METHOD mxGetMk5sData : BOOL
VAR_INPUT
	bItemNumber	: BYTE;
	pstrSetting	: POINTER TO Mk5s_Display_Helpers_Interfaces.strProtectionInfo_v2;
	xSavedData	: BOOL;
END_VAR
VAR_OUTPUT
	bAccesLevelDisplay	: BYTE := _FLAG_Acces_User;
	bAccesLevelEdit	: BYTE := _FLAG_Acces_User;
	xNoEditing	: BOOL := FALSE;
	xNoDisplay	: BOOL := FALSE;
END_VAR
CASE bItemNumber OF
	1:	pstrSetting^.eType := ENUM_VALUE_TYPE.analog;
		pstrSetting^.wTIDName := gTxt_COMITEM_104;
		pstrSetting^.strItem.diValue := itfSTCValve.prpwError;
		xNoDisplay := pstrSetting^.strItem.diValue = 0;
		mxGetMk5sData := TRUE;
ELSE
		mxGetMk5sData := FALSE;
END_CASE
END_METHOD

METHOD mxSetMk5sData : BOOL
VAR_INPUT
	bItemNumber	: BYTE;
	diValue	: DINT;
END_VAR
VAR_OUTPUT
	wSDO	: WORD;
	bSI	: BYTE;
	dataODItem	: Mk5s_Display_Helpers_Interfaces._DEFINITIONS_.ODItem;
	xEditValueSuccessful	: BOOL;
END_VAR
mxSetMk5sData := TRUE;
END_METHOD

METHOD mInit
VAR_INPUT
	itfSTCValveIn	: itf_STCValve;
END_VAR
itfSTCValve := itfSTCValveIn;
END_METHOD

END_FUNCTION_BLOCK

// Aorta/AortaEngine/fbtAortaEngine_Base
FUNCTION_BLOCK fbtAortaEngine_Base IMPLEMENTS itf_STCValve
VAR
	xActive						 : BOOL;
	xActivePI					 : BOOL;	
	bNumberSTC					 : BYTE;
	xCheckCAN					 : BOOL := TRUE;
	xEnergyRecoveryActive		 : BOOL := FALSE;
	itfEnergyRecoveryRegulation  : itf_EnergyRecoveryRegulation;
	bAbsoluteOffset				 : BYTE := 127;
	
	itfIData_PI				: itf_InternalValue_PI;

	fbAorta_Trinamics		: fbtAorta_Trinamics; 
	fbSettingsDownloader 	: fbtAortaSettingsDownloader;
	
	eStateMain				: ENUM_AortaEngine_StateMain;
	eStateHoming			: ENUM_AortaEngine_StateHoming;
	eStateOperating			: ENUM_AortaEngine_StateOperating;
	eStateRetract			: ENUM_AortaEngine_StateRetract;
	
	wEnableErrorCount		: WORD;
	wResetCount				: WORD;
	
	itfLocalRoot			: itf_SystemRoot;
	
	itfWarmUpTemperature		: itf_BaseIO;
	rsWarmUp					: RS;

	itfPositionInput			: itf_BaseIO;
	itfPositionOutput			: itf_BaseIO;
	
	wSDO_STCValve				: WORD;
	
	fbIVL_ActualPosition		: fbtIVL_STCPosition;
	fbIVL_RequiredPosition		: fbtIVL_STCPosition;
	
	fbSTCValve_Protection		: fbtProtecSpec_STCValve;
	
	tFixedPositionTimeoutTime	: TIME;	
	wRangeOffsetLower			: WORD;
	wRangeOffsetUpper			: WORD;
	wWorkingRange				: WORD;
	
	xStart						: BOOL;
	xStartHoming				: BOOL;
	xStartPosition				: BOOL;
	xStartRetract				: BOOL;
	CycleTime 					: TON;

	odError						: ODItem;
	dwStroke_MicroSteps			: DWORD;
	dwStroke_FullSteps			: DWORD;
	rStroke_Rotations			: REAL;
	
	// Settings
	wCycleTime				: WORD;
	wPositioningTimeOut		: WORD;
	wHomingTimeOut			: WORD;

	tInitiateRetryDelayTime		: TIME;
	bMaxHomingRetries			: BYTE;
	bHomingRetries				: BYTE;
	tHomeAgainDelayTime			: TIME;
	tonHomeAgainDelay			: TON;
	dwErrorPosition				: DWORD;
	dwMicroStepsInMove			: DWORD;
	wRetractRange				: WORD;
	wMinimumFullStepRange		: WORD;
	
	diPosition					: DINT;
	dwPositionPrev				: DWORD;
	bFirstWarmUpTemperature		: BYTE;
	wRangeOffsetLowerMargin		: WORD;
	

	iPositionInputRangeMin		: INT;
	iPositionInputRangeMax		: INT;
	iPositionOutputRangeMin		: INT;
	iPositionOutputRangeMax		: INT;
	iPositionOutput				: INT;
	
	itfHomings					: itf_Counter;
    itfStalls					: itf_Counter;
	itfRotations				: itf_Counter;
	
	internalRotationsCounter	: DWORD;
	
	xStartForcedHoming	: BOOL;
	xHomingActive	: BOOL;
	xFixedPositionActive	: BOOL;
	tonFixedPositionTimeout	: TON;

	diPositionInOffState	: DINT;
		
	itfRetainStatus				:itf_Retain_3000_X;
	
	awAlarmNames									: ARRAY[1..6] OF WORD := [gTxt_Alarm_13453, gTxt_Alarm_13454, gTxt_Alarm_13455, gTxt_Alarm_13456, gTxt_Alarm_13457, gTxt_Alarm_13458];
	awAlarmSDOs										: ARRAY[1..6] OF WORD := [16#2815, 16#2895, 16#2896, 16#2897, 16#2898, 16#2899];
	
	awSTCValveHomingCycles							: ARRAY[1..6] OF WORD := [13459, 13460, 13461, 13462, 13463, 13464];
	awSTCValveStalls								: ARRAY[1..6] OF WORD := [13465, 13466, 13467, 13468, 13469, 13470];
	awSTCValveRotations								: ARRAY[1..6] OF WORD := [13471, 13472, 13473, 13474, 13475, 13476];
	
	
	// Debug
	adi_Testing					: ARRAY[1..9] OF DINT;
	diDebugError				: DINT;
	diDebugErrorPosition		: DINT;
	diDebugMicroStepsInMove		: DINT;
	diDebugPosition				: DINT;
	diDebugRotDirection			: DINT;
	diDebugStroke_FullSteps		: DINT;
	diDebugStroke_MicroSteps	: DINT;
	diDebugStroke_Rotations		: DINT;
	diDebugStallDetectPosition	: DINT;
	diDebugStallRetractPosition	: DINT;
	diDebugRetractDelta			: DINT;
	diDebugStatusWord			: DINT;
	diDebugError11Counter		: DINT;
	diDebug_numberStalls		: DINT;
	xDebug_ok					: BOOL;
	wDebugError2				: WORD;

END_VAR

METHOD mxInit_SysPyLog : BOOL
VAR_INPUT
END_VAR
SysPyLog.mxAdd(eCode := eLogCodes._fixed_1, pData := ADR(xDebug_ok),sNaam := 'xOk', eType := eLogTypes._byte);
SysPyLog.mxAdd(eCode := eLogCodes._fixed_1, pData := ADR(odError.wValue[1]),sNaam := 'Aorta Error', eType := eLogTypes._word);
SysPyLog.mxAdd(eCode := eLogCodes._fixed_1, pData := ADR(wDebugError2),sNaam := 'Aorta Error2', eType := eLogTypes._word);
SysPyLog.mxAdd(eCode := eLogCodes._fixed_1, pData := ADR(eStateMain),sNaam := 'State Main', eType := eLogTypes._byte);
SysPyLog.mxAdd(eCode := eLogCodes._fixed_1, pData := ADR(eStateOperating),sNaam := 'State Operating', eType := eLogTypes._byte);
SysPyLog.mxAdd(eCode := eLogCodes._fixed_1, pData := ADR(eStateHoming),sNaam := 'State Homing', eType := eLogTypes._byte);
SysPyLog.mxAdd(eCode := eLogCodes._fixed_1, pData := ADR(diDebugStroke_FullSteps),sNaam := 'Full steps stroke', eType := eLogTypes._byte);
SysPyLog.mxAdd(eCode := eLogCodes._fixed_1, pData := ADR(diDebugErrorPosition),sNaam := 'Error Position', eType := eLogTypes._dint);
SysPyLog.mxAdd(eCode := eLogCodes._fixed_1, pData := ADR(diDebugMicroStepsInMove),sNaam := 'Micro Steps In Move', eType := eLogTypes._dint);
SysPyLog.mxAdd(eCode := eLogCodes._fixed_1, pData := ADR(diDebugRotDirection),sNaam := 'Rotation Direction', eType := eLogTypes._dint);
SysPyLog.mxAdd(eCode := eLogCodes._fixed_1, pData := ADR(diDebugStroke_FullSteps),sNaam := 'Stroke In Full Steps', eType := eLogTypes._dint);
SysPyLog.mxAdd(eCode := eLogCodes._fixed_1, pData := ADR(diDebug_numberStalls),sNaam := 'Number of Stalls', eType := eLogTypes._dint);
END_METHOD

METHOD mxInit : BOOL
VAR_INPUT
	wSDOIn			: WORD;
	itfEnergyRecoveryRegulationIn : itf_EnergyRecoveryRegulation;
END_VAR
VAR
	TmpItem	: ODItem;		
	itfLookupTables	: itf_lookuptables;
	itfCounters		: itf_Counters;
END_VAR
mxInit := TRUE;
xActive := TRUE;

IF NOT __QUERYINTERFACE(GVL_itfRoot,	itfLocalRoot) THEN	mxInit := FALSE;	RETURN;	END_IF

IF NOT CmpODRead(wSDO_STCValve,	27,	ADR(TmpItem))  THEN
	xActive := FALSE;
	fbIVL_ActualPosition.prpxDataBaseDefined 	:= FALSE;
	fbIVL_RequiredPosition.prpxDataBaseDefined  := FALSE;
	RETURN;
END_IF

IF TmpItem.bValue[3] = 0 THEN
	xActive := FALSE;
END_IF

itfCounters					:= itfLocalRoot.prpitfCounters;
itfLocalRoot.prpitfRetain.mxGetRetainPrimaryMachine(itfRetainPrimaryMachineStatus=>itfRetainStatus);
itfLocalRoot.prpitfCANtainer.mxAttachDriver(eType := eTypeDrivers.AortaDrives, itfcanopendriver := fbAorta_Trinamics.prpitfCANOpenDriver);
itfLocalRoot.prpitfCANtainer.mxAttachDownloader(itfsettingsdownloader := fbSettingsDownloader);
itfLookupTables				:= itfLocalRoot.prpitfLookupTables;

IF		itfLookupTables	= 0 OR	itfCounters	= 0 OR itfRetainStatus = 0 THEN	
	mxInit := FALSE;	RETURN;	END_IF

itfHomings		:= itfCounters.mitfGetCounter(awSTCValveHomingCycles[bNumberSTC]);
itfStalls		:= itfCounters.mitfGetCounter(awSTCValveStalls[bNumberSTC]);
itfRotations	:= itfCounters.mitfGetCounter(awSTCValveRotations[bNumberSTC]);

mxInit := mxInit AND mxLoadSettings(itfEnergyRecoveryRegulationIn); 

xStart := TRUE;
eStateMain := ENUM_AortaEngine_StateMain.Enable;
wEnableErrorCount := 0;
wResetCount := 0;

fbAorta_Trinamics.mxInit(bCANAddress := 6 ,wHomingTimeOutIn := wHomingTimeOut ,wPositioningTimeOutIn :=wPositioningTimeOut );
fbSettingsDownloader.mxInit(ADR(fbAorta_Trinamics));

// Initialising STC Valve Alarm
mxInit := mxInit AND fbSTCValve_Protection.mxInitSpecial(wNameIn := awAlarmNames[bNumberSTC], wSDOIn := awAlarmSDOs[bNumberSTC], THIS^);

mxInit_SysPyLog();
END_METHOD

METHOD mxInit_Output : BOOL
VAR_INPUT
	bNumberSTCIn			: BYTE;
	wSDOIn					: WORD;
	wMPL_actualPosition		: WORD;
	wMPL_requiredPosition	: WORD;
	wName_actualPosition	: WORD;
	wName_requiredPosition	: WORD;
END_VAR
VAR
	itfLookupTables	: itf_lookuptables;
END_VAR
mxInit_Output := TRUE;
bNumberSTC := bNumberSTCIn;
wSDO_STCValve := wSDOIn;
mxInit_Output := mxInit_Output AND fbIVL_ActualPosition.mxInit(wMPL_actualPosition);
mxInit_Output := mxInit_Output AND fbIVL_RequiredPosition.mxInit(wMPL_requiredPosition);
END_METHOD

METHOD mxLoadSettings : BOOL
VAR_INPUT
	itfEnergyRecoveryRegulationIn : itf_EnergyRecoveryRegulation;
END_VAR
VAR
	TmpItem						  : ODItem;
	tFixedPositionTimeoutTimeUnit : ENUM_TimeUnit;
	i							  : BYTE;
	itfIData_temp				  : itf_InternalValue;
END_VAR
// Collect Data
mxLoadSettings := TRUE;

FOR i := 1 TO 11 BY 1 DO //see Hi5 SDO 2666
    CmpODRead(ENUM_SDO_2000.Aorta, i ,ADR(TmpItem));

	CASE i OF
		
	1: 
		tInitiateRetryDelayTime		:= TmpItem.bValue[1] * T#1S;
		bMaxHomingRetries			:= TmpItem.bValue[2];
		tHomeAgainDelayTime			:= TmpItem.bValue[3] * T#1H;
		wHomingTimeOut 				:= TmpItem.bValue[4];
	
	2:
		wRetractRange			:= TmpItem.wValue[1];
		wMinimumFullStepRange	:= TmpItem.wValue[2];
	
	3:
	
		wRangeOffsetLower	:= TmpItem.wValue[1];
		wCycleTime 			:= TmpItem.wValue[2];
		
	4:
		wPositioningTimeOut := TmpItem.wValue[1];
		IF TmpItem.wValue[2] = 0 THEN mxLoadSettings:= FALSE; RETURN; END_IF; 
		itfLocalRoot.prpitfLookupTables.prpitfIVLList.mxFind(wFind:=TmpItem.wValue[2], itfFound=>itfIData_temp);  
		IF NOT __QUERYINTERFACE(itfIData_temp,	itfIData_PI) THEN	mxLoadSettings := FALSE;	RETURN;	END_IF 
		mxLoadSettings:=mxLoadSettings AND itfIData_PI<>0;
		
	5:
		wRangeOffsetUpper	:= GVL_Aorta.wControlRange - TmpItem.wValue[1];
		IF itfPositionOutput <> 0 THEN
			itfLocalRoot.prpitfLookupTables.prpitfMPLList.mxFind(wFind:=TmpItem.wValue[2], itfFound=>itfPositionOutput);
			mxLoadSettings:=mxLoadSettings AND itfPositionOutput<>0;	
		END_IF
		
			
	9:
		wRangeOffsetLowerMargin	:= TmpItem.wValue[1];
		bFirstWarmUpTemperature	:= TmpItem.bValue[3];
	
	10:
		IF TmpItem.wValue[2] <> 0 THEN
			itfLocalRoot.prpitfLookupTables.prpitfMPLList.mxFind(wFind:=TmpItem.wValue[2], itfFound=>itfPositionInput);
			mxLoadSettings:=mxLoadSettings AND itfPositionInput<>0;
		END_IF
		
		
	11:
		IF TmpItem.wValue[1] = 0 THEN mxLoadSettings:= FALSE; RETURN; END_IF; 
		itfLocalRoot.prpitfLookupTables.prpitfMPLList.mxFind(wFind:=TmpItem.wValue[1], itfFound=>itfWarmUpTemperature);
		mxLoadSettings:=mxLoadSettings AND itfWarmUpTemperature<>0;

	ELSE
		IF NOT (i = 6 OR i = 7 OR i = 8) THEN
			mxLoadSettings := FALSE;	
		END_IF
	END_CASE
END_FOR

CmpODRead(ENUM_SDO_2000.Aorta,	23,	ADR(TmpItem));
tFixedPositionTimeoutTimeUnit := TmpItem.bValue[3];
xEnergyRecoveryActive		  := BYTE_TO_BOOL(TmpItem.bValue[2]);

CASE tFixedPositionTimeoutTimeUnit OF
	ENUM_TimeUnit.Millisecond	: tFixedPositionTimeoutTime := TmpItem.bValue[4] * T#1MS;
	ENUM_TimeUnit.Second	: tFixedPositionTimeoutTime := TmpItem.bValue[4] * T#1S;
	ENUM_TimeUnit.Minute	: tFixedPositionTimeoutTime := TmpItem.bValue[4] * T#1M;
	ENUM_TimeUnit.Hour	: tFixedPositionTimeoutTime := TmpItem.bValue[4] * T#1H;
	ENUM_TimeUnit.Day	: tFixedPositionTimeoutTime := TmpItem.bValue[4] * T#1D;
END_CASE

wWorkingRange	:= wRangeOffsetUpper - wRangeOffsetLower;

IF xEnergyRecoveryActive = 1 THEN
	mxLoadSettings := mxLoadSettings AND CmpODRead(_wSDO2_EnergyRecoveryRegulation, 1, ADR(TmpItem));
	itfEnergyRecoveryRegulation := itfEnergyRecoveryRegulationIn;
	mxLoadSettings := mxLoadSettings AND itfEnergyRecoveryRegulation <> 0;
END_IF

CmpODRead(ENUM_SDO_2000.Aorta,	35,	ADR(TmpItem));	
	diPositionInOffState:=TmpItem.diValue;
END_METHOD

METHOD mxRun : BOOL
VAR
	wError	: WORD;
	bError  : BYTE;
	xOk		: BOOL;
	xSwitchToER		: BOOL;
END_VAR
IF NOT xActive THEN
	RETURN;
END_IF

//  fbAorta_Trinamics.mxRun(); running via CANTainer
IF (fbAorta_Trinamics.mxConfigurationError(bError => bError) OR THIS^.prpxCANDriverError) AND xCheckCAN THEN
	eStateMain	:= ENUM_AortaEngine_StateMain.CAN_Error;
	xCheckCAN := FALSE;
END_IF

fbIVL_ActualPosition.mxSetOutput(TO_REAL(fbAorta_Trinamics.prpdwPosition));
fbIVL_RequiredPosition.mxSetOutput(TO_REAL(fbAorta_Trinamics.prpdwRequiredPosition));

IF eStateMain <> ENUM_AortaEngine_StateMain.Operating THEN 
	xActivePI := FALSE;
	itfIData_PI.prpxActiveSTCPIRegulation := xActivePI;
END_IF

CASE eStateMain OF	

	ENUM_AortaEngine_StateMain.Enable :
		IF	mxEnable(xStart := xStart, xOk => xOk,  wError => wError)	THEN
			IF	xOk	THEN
				eStateMain	:= ENUM_AortaEngine_StateMain.Homing;
				xStart := TRUE;
 				wEnableErrorCount := 0;
 			ELSE
				IF wEnableErrorCount > 1 THEN
	 				THIS^.odError.wValue[1] := wError;
					eStateMain := ENUM_AortaEngine_StateMain.Error;
				ELSE
					wEnableErrorCount := wEnableErrorCount + 1; 
					eStateMain	:= ENUM_AortaEngine_StateMain.Reset;
					wResetCount := 0;
				END_IF
			END_IF
		END_IF
		
	ENUM_AortaEngine_StateMain.Reset : 
		CASE  wResetCount OF
		 0 : 	fbAorta_Trinamics.prpitfCANOpenDriver.mxReset();
		 5 :  	fbAorta_Trinamics.prpitfCANOpenDriver.mxStart();
		 50:	xStart := TRUE;
		 		IF fbAorta_Trinamics.mxConfigurationError(bError => bError) THEN
					THIS^.odError.wValue[1] := bError + 256;
					eStateMain	:= ENUM_AortaEngine_StateMain.Error;
				ELSIF THIS^.prpxCANDriverError THEN
					THIS^.odError.wValue[1] := Aorta_Errors.CAN_Out;
					eStateMain	:= ENUM_AortaEngine_StateMain.Error;
				ELSE
					eStateMain	:= ENUM_AortaEngine_StateMain.Enable;
					xCheckCAN	:= TRUE;
				END_IF				 
		END_CASE
		wResetCount := wResetCount + 1;

	ENUM_AortaEngine_StateMain.Homing :
		xHomingActive := TRUE;
		xStartForcedHoming := FALSE;
		IF	mxHoming(xStart := xStart , xOk => xOk, wError => wError) THEN
			IF xOk THEN
				itfHomings.mIncrement();
				tonHomeAgainDelay(IN := FALSE);
				bHomingRetries := 0;
				eStateMain	:= ENUM_AortaEngine_StateMain.Operating;
				xStart := TRUE;
				xHomingActive := FALSE;
			ELSE
				IF	bHomingRetries < bMaxHomingRetries	THEN
					bHomingRetries	:= bHomingRetries + 1;
					eStateMain	:= ENUM_AortaEngine_StateMain.Homing;
					xStart			:= TRUE;				
				ELSE
					THIS^.odError.wValue[1]	:= wError;
					// where to go?
					// FV: add stopped/alarm status that only can exit via warning reset
					eStateMain	:= ENUM_AortaEngine_StateMain.Error;
					xStart := TRUE;
				END_IF
			END_IF
		END_IF
		
	ENUM_AortaEngine_StateMain.Operating :

		tonHomeAgainDelay(IN := tHomeAgainDelayTime <> T#0H, PT := tHomeAgainDelayTime);
		IF	mxOperating(xStart := xStart, xOk => xOk, wError => wError)	THEN
			IF xOk THEN 
				IF	(tonHomeAgainDelay.Q AND itfRetainStatus.prpw_xS <> _STATEINFO_wCS2090_Shutdown) OR xStartForcedHoming	THEN
					eStateMain	:= ENUM_AortaEngine_StateMain.Homing;
				END_IF
				xStart := TRUE;
			ELSE
 				THIS^.odError.wValue[1]	:= wError;
				IF wError = Aorta_Errors.Position_Stall THEN
					eStateMain := ENUM_AortaEngine_StateMain.Retract;
					xStart := TRUE;
				ELSE
					eStateMain	:= ENUM_AortaEngine_StateMain.Error;
					xStart := TRUE;
				END_IF
			END_IF
		END_IF

	ENUM_AortaEngine_StateMain.Retract :

		IF	mxRetract(xStart := xStart, xOk => xOk, wError => wError)	THEN
			itfStalls.mIncrement();
			IF xOk THEN 
				eStateMain	:= ENUM_AortaEngine_StateMain.Operating;
				xStart := TRUE;
			ELSE
				eStateMain	:= ENUM_AortaEngine_StateMain.Homing;
				xStart 		:= TRUE;
 				THIS^.odError.wValue[1]	:= wError;
			END_IF
		END_IF
		
	ENUM_AortaEngine_StateMain.Error :
		fbAorta_Trinamics.mxDisable(xStart:=xStart);
		IF THIS^.odError.wValue[1] = 0 THEN
			THIS^.odError.wValue[1] := Aorta_Errors.StuckInErrorState;
		END_IF
		
	ENUM_AortaEngine_StateMain.CAN_Error :
		wResetCount := 0;
		eStateMain := ENUM_AortaEngine_StateMain.Reset;
	
	// Only used for debugging, put xStart manually on true and change eStateMain to Valve detached.
	ENUM_AortaEngine_StateMain.Valve_detached :  
		IF fbAorta_Trinamics.mxPosition( xStart := xStart, dwPosition := TO_DWORD(-5000), xRelative := TRUE, xok => xok) THEN	
			IF xOk THEN 
				eStateMain	:= ENUM_AortaEngine_StateMain.Enable;
				xStart := TRUE;
			ELSE
				eStateMain	:= ENUM_AortaEngine_StateMain.Error;
				xStart := TRUE;
			END_IF
		END_IF	
	
END_CASE 

// Debugging

diDebugError				:= TO_DINT(THIS^.odError.wValue[1]); // ok
wDebugError2				:= wError;
diDebugErrorPosition		:= TO_DINT(dwErrorPosition);
diDebugMicroStepsInMove		:= TO_DINT(dwMicroStepsInMove);
diDebugPosition				:= TO_DINT(fbAorta_Trinamics.prpdwPosition);
diDebugRotDirection			:= TO_DINT(fbAorta_Trinamics.prpxDirection);
diDebugStroke_FullSteps		:= TO_DINT(dwStroke_FullSteps);
diDebugStroke_MicroSteps	:= TO_DINT(dwStroke_MicroSteps);
diDebugStroke_Rotations		:= TO_DINT(rStroke_Rotations);
diDebugStatusWord			:= TO_DINT(fbAorta_Trinamics.prpwSW);
diDebugError11Counter		:= TO_DINT(fbAorta_Trinamics.prpdwError11Count);
diDebug_numberStalls		:= TO_DINT(itfStalls.prpdwValue);
xDebug_ok					:=xOk;

mxCollectInfoSDO3000(bIndex := 1, diInput := THIS^.odError.wValue[1]);
mxCollectInfoSDO3000(bIndex := 2, diInput := TO_DINT(fbAorta_Trinamics.prpxDirection));
mxCollectInfoSDO3000(bIndex := 3, diInput := TO_DINT(fbAorta_Trinamics.prpdwPosition));
mxCollectInfoSDO3000(bIndex := 4, diInput := TO_DINT(fbAorta_Trinamics.prpdwRequiredPosition));
mxCollectInfoSDO3000(bIndex := 5, diInput := TO_DINT(dwStroke_FullSteps));
mxCollectInfoSDO3000(bIndex := 6, diInput := TO_DINT(fbAorta_Trinamics.prpwSW));
mxCollectInfoSDO3000(bIndex := 7, diInput := TO_DINT(itfStalls.prpdwValue));
mxCollectInfoSDO3000(bIndex := 8, diInput := TO_DINT(itfHomings.prpdwValue));
IF itfEnergyRecoveryRegulation <> 0 THEN
	 xSwitchToER := itfEnergyRecoveryRegulation.prpxSwitchToER;
END_IF
mxCollectInfoSDO3000(bIndex := 9, diInput := TO_DINT(xSwitchToER));

IF itfPositionOutput <> 0 THEN
	iPositionOutput := TO_INT(fdintLinearInterpolation(0, iPositionOutputRangeMin, GVL_Aorta.wControlRange, iPositionOutputRangeMax, TO_INT(fbAorta_Trinamics.prpdwPosition)));
	itfPositionOutput.mxSetValueInt(iPositionOutput, FALSE);
END_IF
END_METHOD

METHOD PRIVATE mxHoming : BOOL
VAR_IN_OUT
	xStart : BOOL;
END_VAR
VAR_OUTPUT
	wError	: WORD;
	xOk		: BOOL;
END_VAR
IF xStart THEN
	xStartHoming := TRUE;
	eStateHoming := ENUM_AortaEngine_StateHoming.Home;
	xStart := FALSE;
END_IF

CASE eStateHoming OF

	ENUM_AortaEngine_StateHoming.Home :
		IF	fbAorta_Trinamics.mxHoming(	xStart				:= xStartHoming,
										dwStroke_microSteps	=> dwStroke_MicroSteps,
										dwStroke_FullSteps	=> dwStroke_FullSteps,
										rRotations			=> rStroke_Rotations,
										xOk					=> xOk,
										wError				=> wError)	THEN
			IF	xOk	THEN
				eStateHoming	:= ENUM_AortaEngine_StateHoming.CheckRange;
			ELSE
				mxHoming		:= TRUE;
			END_IF
		END_IF
	
	ENUM_AortaEngine_StateHoming.CheckRange :
		IF	dwStroke_FullSteps < wMinimumFullStepRange	THEN
			wError			:= Aorta_Errors.Homing_RangeTooSmall;
			xOk 			:= FALSE;
		ELSE
			xOk := TRUE;
		END_IF
		mxHoming	:= TRUE;
END_CASE
END_METHOD

METHOD PRIVATE mxOperating : BOOL
VAR_IN_OUT
	xStart : BOOL;
END_VAR
VAR_OUTPUT
	wError	: WORD;
	xOk     : BOOL;
END_VAR
VAR
	dwMicroStepsInMove	: DWORD;
	xActivePIRegulation	: BOOL;
	xSwitchToER			: BOOL;
END_VAR
IF xStart THEN
	eStateOperating := ENUM_AortaEngine_StateOperating.SetNextPosition;
	xStart := FALSE;
END_IF

IF itfEnergyRecoveryRegulation <> 0 THEN
	 xSwitchToER := itfEnergyRecoveryRegulation.prpxSwitchToER;
END_IF

itfIData_PI.prpxActiveSTCPIRegulation := xActivePI;


CASE eStateOperating OF
	
	ENUM_AortaEngine_StateOperating.SetNextPosition :
		IF NOT xFixedPositionActive AND itfRetainStatus.prpw_xS = _STATEINFO_wCS2020_Off OR
 (NOT xFixedPositionActive AND xEnergyRecoveryActive AND NOT xSwitchToER)THEN 
			diPosition:=diPositionInOffState;
			xActivePI := FALSE;
			
		ELSIF NOT xFixedPositionActive THEN // Position set in mxMoveToFixedPosition
			tonFixedPositionTimeout(IN := FALSE, PT := tFixedPositionTimeoutTime);
			dwPositionPrev := fbAorta_Trinamics.prpdwPosition;	
			IF itfPositionInput <> 0 AND_THEN NOT itfPositionInput.prpxSensorError THEN // Position via 4-20mA
				itfPositionInput.mxGetValueINT(iValueOut => diPosition);
				diPosition := fdintLinearInterpolation(iPositionInputRangeMin, 0, iPositionInputRangeMax, GVL_Aorta.wControlRange, diPosition);
				xActivePI := FALSE;
			ELSE // Position via algorithm
				IF itfIData_PI.prpxSensorError THEN
					wError := Aorta_Errors.Position_PI_Error;
					xActivePI := FALSE;
				ELSE
					diPosition := mdiNextPosition(TO_DINT(dwPositionPrev));
					xActivePI := TRUE;
				END_IF
				
			END_IF			
		ELSE
			// Run timer to turn off xFixedPositionActive
			xActivePI := FALSE;
			tonFixedPositionTimeout(IN := TRUE, PT := tFixedPositionTimeoutTime);
			IF tonFixedPositionTimeout.Q THEN
				tonFixedPositionTimeout(IN := FALSE, PT := tFixedPositionTimeoutTime);
				xFixedPositionActive := FALSE;
			END_IF
		END_IF

		diPosition	:= LIMIT(wRangeOffsetLower, diPosition, wRangeOffsetUpper);
		xStartPosition := TRUE;
		eStateOperating := ENUM_AortaEngine_StateOperating.GoToPosition;
		
	ENUM_AortaEngine_StateOperating.GoToPosition	:

		IF fbAorta_Trinamics.mxPosition( xStart := xStartPosition, dwPosition := TO_DWORD(diPosition), xRelative := FALSE, xOk => xOk,wError => wError, dwMicroStepsInMove => dwMicroStepsInMove) THEN
			IF xOk THEN
				THIS^.dwMicroStepsInMove := dwMicroStepsInMove;
				eStateOperating := ENUM_AortaEngine_StateOperating.Wait;
				CycleTime(IN:=FALSE,PT:= wCycleTime * T#1MS);
			ELSE
				mxOperating	:= TRUE;
			END_IF
			internalRotationsCounter := internalRotationsCounter + (ABS(dwPositionPrev - fbAorta_Trinamics.prpdwPosition) * dwStroke_MicroSteps / GVL_Aorta.wControlRange);
			IF internalRotationsCounter >= 51200 THEN
				itfRotations.mIncrement();
				internalRotationsCounter := internalRotationsCounter - 51200;
			END_IF
		END_IF
		
	ENUM_AortaEngine_StateOperating.Wait :
	
		CycleTime(IN:=TRUE,PT:= wCycleTime * T#1MS);
		IF CycleTime.Q THEN
			eStateOperating := ENUM_AortaEngine_StateOperating.SetNextPosition;
			xOK:=TRUE;
			mxOperating:=TRUE;
		END_IF;

END_CASE
END_METHOD

METHOD PRIVATE mxEnable : BOOL
VAR_IN_OUT
	xStart : BOOL;
END_VAR
VAR_OUTPUT
	xOk 	: BOOL;
	wError 	: WORD;
END_VAR
mxEnable := fbAorta_Trinamics.mxEnable(	xStart	:= xStart, xOk => xOk, wError	=> wError);
END_METHOD

METHOD PRIVATE mxRetract : BOOL
VAR_IN_OUT
	xStart : BOOL;
END_VAR
VAR_OUTPUT
	wError	: WORD;
	xOk		: BOOL;
END_VAR
VAR
	diDelta : DINT;
	dwActualPosition : DWORD;
END_VAR
IF xStart THEN
	eStateRetract := ENUM_AortaEngine_StateRetract.SetRetractPosition;
	xStart := FALSE;
END_IF

CASE eStateRetract OF
	
	ENUM_AortaEngine_StateRetract.SetRetractPosition :

		dwActualPosition := fbAorta_Trinamics.prpdwPosition;	
		diDelta	:= SEL(fbAorta_Trinamics.prpxDirection, 1, -1) * WORD_TO_INT(wRetractRange);
		diPosition	:= TO_DINT(dwActualPosition) + diDelta;
		diPosition	:= LIMIT(0, diPosition, GVL_Aorta.wControlRange);

		
		diDebugStallDetectPosition := DWORD_TO_DINT(dwActualPosition);
		diDebugStallRetractPosition := diPosition;
		diDebugRetractDelta := diDelta;

		
		xStartRetract := TRUE;
		eStateRetract := ENUM_AortaEngine_StateRetract.Retract;

	ENUM_AortaEngine_StateRetract.Retract :

		IF fbAorta_Trinamics.mxPosition( xStart := xStartRetract, dwPosition := TO_DWORD(diPosition),xRelative := FALSE, xOk => xOk,wError => wError, dwMicroStepsInMove => dwMicroStepsInMove) THEN
			IF xOk THEN
				mxRetract		:= TRUE;
				wError			:= Aorta_Errors.NoError;
			ELSE
				mxRetract		:= TRUE;
				wError			:= Aorta_Errors.Position_Retract;
			END_IF
		END_IF
		
END_CASE
END_METHOD

METHOD mdiNextPosition : DINT
VAR_INPUT
	diCurrentPosition	: DINT;
END_VAR
VAR_OUTPUT
END_VAR
VAR
	iActualTemperature	: INT;
	dideltaPosition		: DINT;
END_VAR
IF bFirstWarmUpTemperature > 0 THEN
	itfWarmUpTemperature.mxGetValueINT(iValueOut => iActualTemperature);
END_IF
rsWarmUp(SET := dwPositionPrev <= wRangeOffsetLower + wRangeOffsetLowerMargin, RESET1 := iActualTemperature >= bFirstWarmUpTemperature * 10);
IF NOT rsWarmUp.Q1 THEN
	itfIData_PI.mxGetValueDINT( diValueOut => dideltaPosition);
	mdiNextPosition := diCurrentPosition + dideltaPosition;
ELSE
	mdiNextPosition := 0;
END_IF
END_METHOD

PROPERTY prppdiDebugPosition : POINTER TO DINT
GET
prppdiDebugPosition := ADR(diDebugPosition);
END_GET
END_PROPERTY

PROPERTY prppdiDebugStroke_FullSteps : POINTER TO DINT
GET
prppdiDebugStroke_FullSteps := ADR(diDebugStroke_FullSteps);
END_GET
END_PROPERTY

PROPERTY prppdiDebugStroke_MicroSteps : POINTER TO DINT
GET
prppdiDebugStroke_MicroSteps := ADR(diDebugStroke_MicroSteps);
END_GET
END_PROPERTY

PROPERTY prppdiDebugStroke_Rotations : POINTER TO DINT
GET
prppdiDebugStroke_Rotations := ADR(diDebugStroke_Rotations);
END_GET
END_PROPERTY

PROPERTY prppdiDebugError : POINTER TO DINT
GET
prppdiDebugError := ADR(diDebugError);
END_GET
END_PROPERTY

PROPERTY prppdiDebugErrorPosition : POINTER TO DINT
GET
prppdiDebugErrorPosition := ADR(diDebugErrorPosition);
END_GET
END_PROPERTY

PROPERTY prppdiDebugMicroStepsInMove : POINTER TO DINT
GET
prppdiDebugMicroStepsInMove := ADR(diDebugMicroStepsInMove);
END_GET
END_PROPERTY

PROPERTY prppdiDebugRotDirection : POINTER TO DINT
GET
prppdiDebugRotDirection := ADR(diDebugRotDirection);
END_GET
END_PROPERTY

PROPERTY prppdiDebugStallDetectPosition : POINTER TO DINT
GET
prppdiDebugStallDetectPosition := ADR(diDebugStallDetectPosition);
END_GET
END_PROPERTY

PROPERTY prppdiDebugStallRetractDelta : POINTER TO DINT
GET
prppdiDebugStallRetractDelta := ADR(diDebugRetractDelta);
END_GET
END_PROPERTY

PROPERTY prppdiDebugStallRetractPosition : POINTER TO DINT
GET
prppdiDebugStallRetractPosition := ADR(diDebugStallRetractPosition);
END_GET
END_PROPERTY

PROPERTY prppdiStatusWord : POINTER TO DINT
GET
prppdiStatusWord := ADR(diDebugStatusWord);
END_GET
END_PROPERTY

PROPERTY prppdiDebugError11Counter : POINTER TO DINT
GET
prppdiDebugError11Counter:=ADR(diDebugError11Counter);
END_GET
END_PROPERTY

PROPERTY prpdwPosition : DWORD
GET
prpdwPosition := fbAorta_Trinamics.prpdwPosition;
END_GET
END_PROPERTY

PROPERTY prpwError : WORD
GET
PUBLIC 
VAR
END_VAR
prpwError := odError.wValue[1];
END_GET
SET
PUBLIC 
VAR
END_VAR
odError.wValue[1] := prpwError;
END_SET
END_PROPERTY

METHOD mReset
eStateMain	:= ENUM_AortaEngine_StateMain.Enable;
wEnableErrorCount := 0;
wResetCount := 0;
odError.wValue[1] := 0;
bHomingRetries := 0;
xStart := TRUE;
END_METHOD

METHOD mxOD3000Define : BOOL
VAR_INPUT
	itf0D3000 		: itf_od3000;
	awSDO			: ARRAY[1..6] OF WORD;
END_VAR
VAR
	Data		: _OD3000Struct_RegistrationData;
	i			: BYTE;
	j			: DINT;
	bOffset		: BYTE;
END_VAR
mxOD3000Define:=TRUE;

IF xActive THEN
	// Find correct Transformation dataset 
	FOR j := LOWER_BOUND(awSDO, 1) TO UPPER_BOUND(awSDO, 1) DO
		IF awSDO[j] = wSDO_STCValve THEN
			bOffset := (DINT_TO_BYTE(j)-1)*TO_BYTE(SIZEOF(adi_Testing));
		END_IF
	END_FOR
	
	// Define SDO 3000
	FOR i := 1 TO TO_BYTE(SIZEOF(adi_Testing)) DO
		Data.wIndex		:= _wSDO3_STC_oilfree_Testing;
		Data.bSubIndex	:= i + bOffset + bAbsoluteOffset;										 
		Data.pData		:= ADR(adi_Testing[i]);
		Data.wAttrib	:= _OD3000_wSubIndexRead;
		mxOD3000Define	:= mxOD3000Define AND itf0D3000.mxAdd(Data);
	END_FOR
END_IF
END_METHOD

METHOD mxConfigurationError : BOOL
VAR_OUTPUT
	bError : BYTE;
END_VAR
mxConfigurationError := fbAorta_Trinamics.mxConfigurationError(bError => bError);
END_METHOD

PROPERTY prprLimitedPosition : REAL
GET
// prpdwLimitedPosition := (prpdwPosition - wRangeOffsetLower) / (wRangeOffsetUpper - wRangeOffsetLower) * 100;

prprLimitedPosition := TO_REAL(prpdwPosition - wRangeOffsetLower) / TO_REAL(wWorkingRange);
END_GET
END_PROPERTY

PROPERTY prpxActive : BOOL
GET
prpxActive := xActive;
END_GET
END_PROPERTY

PROPERTY prpxFixedPositionActive : BOOL
GET
prpxFixedPositionActive := xFixedPositionActive;
END_GET
END_PROPERTY

PROPERTY prpxHomingActive : BOOL
GET
prpxHomingActive := xHomingActive;
END_GET
END_PROPERTY

METHOD mxStartHoming : BOOL
IF NOT xHomingActive THEN
	xStartForcedHoming := TRUE;
END_IF
END_METHOD

METHOD mxMoveToFixedPosition : BOOL
VAR_INPUT
	dwPosition	: DWORD;
END_VAR
xFixedPositionActive := TRUE;
diPosition := TO_DINT(dwPosition);
END_METHOD

PROPERTY prpdwHomingStrokeMS : DWORD
GET
prpdwHomingStrokeMS:=dwStroke_MicroSteps;
END_GET
END_PROPERTY

PROPERTY prpxCANDriverError : BOOL
GET
prpxCANDriverError := fbAorta_Trinamics.prpitfCANOpenDriver.prpxIsNotOK;
END_GET
END_PROPERTY

METHOD mxCollectInfoSDO3000 : BOOL
VAR_INPUT
	bIndex	: BYTE;
	diInput	: DINT;
END_VAR
mxCollectInfoSDO3000 := TRUE;
// Check index
IF bIndex <= 0 OR bIndex > TO_BYTE(SIZEOF(adi_Testing)) THEN
	mxCollectInfoSDO3000 := FALSE;
	RETURN;
END_IF

adi_Testing[bIndex]:=diInput;
END_METHOD

END_FUNCTION_BLOCK

// Aorta/AortaEngine/IVL/fbtIVL_STCPosition
FUNCTION_BLOCK fbtIVL_STCPosition EXTENDS fbtIVL_OutputBase
VAR
END_VAR

(*Stijn Staring - 05/04/2023*)

METHOD mxIVL_Settings_Overwrite : BOOL
VAR_INPUT
	wIVL_number	: WORD;
END_VAR
fbIVL_Out.mxInit(0, wIVL_number, _IVL_bAnalogType_Percent_001);
END_METHOD

END_FUNCTION_BLOCK

// Aorta/Driver/CANOpenDriver/PDO Topic/Rx/fbtAorta_ActualPosition_1
FUNCTION_BLOCK fbtAorta_ActualPosition_1 EXTENDS fbtPDO_DWORD
VAR_INPUT
END_VAR
VAR_OUTPUT
END_VAR
VAR
//	dwPosition : DWORD;
END_VAR

PROPERTY prpdwPosition : DWORD
GET
prpdwPosition:=dwData;
END_GET
END_PROPERTY

END_FUNCTION_BLOCK

// Oil Free Air/Offset/fbtOffsetsConditionalSetpointCalculation
FUNCTION_BLOCK fbtOffsetsConditionalSetpointCalculation IMPLEMENTS itf_OffsetsConditionalSetpointCalculation
VAR
	xActive											: BOOL := FALSE;
	bAmountOffsets									: BYTE := 8;
	
	fbOffset1										: fbtOffset;
	fbOffset2										: fbtOffset;
	fbOffset3										: fbtOffset;
	fbOffset4										: fbtOffset;
	fbOffset5										: fbtOffset;
	fbOffset6										: fbtOffset;
	fbOffset7										: fbtOffset;
	fbOffset8										: fbtOffset;
	
	//Testing
	adi_Testing		: ARRAY[1..8] OF DINT; // [diOffset1, ... , diOffset8]

END_VAR

(*
Stijn Staring - 31/03/23
This offset function should be used together with the Conditional Setpoint Calculation functions.
In the Conditional Setpoint Calculation functions there will be options provided to apply the offset. 

Options =>
•	Absolute offset: the obvious; add or substract the given value
•	IData
•	MPL

Safety value to detect a sensor error.
*)

METHOD mxInit : BOOL
VAR_INPUT
END_VAR
VAR
	TmpItem		: ODItem;
END_VAR
mxInit:=TRUE;
xActive:=TRUE;

IF NOT CmpODRead(_wSDO2_OffsetsConditionalSetpoint, 1 ,ADR(TmpItem)) THEN
	xActive:=FALSE;
	RETURN;
END_IF

mxInit:= mxInit AND fbOffset1.mxInit(1,_wSDO2_OffsetsConditionalSetpoint);
mxInit:= mxInit AND fbOffset2.mxInit(2,_wSDO2_OffsetsConditionalSetpoint);
mxInit:= mxInit AND fbOffset3.mxInit(3,_wSDO2_OffsetsConditionalSetpoint);
mxInit:= mxInit AND fbOffset4.mxInit(4,_wSDO2_OffsetsConditionalSetpoint);
mxInit:= mxInit AND fbOffset5.mxInit(5,_wSDO2_OffsetsConditionalSetpoint);
mxInit:= mxInit AND fbOffset6.mxInit(6,_wSDO2_OffsetsConditionalSetpoint);
mxInit:= mxInit AND fbOffset7.mxInit(7,_wSDO2_OffsetsConditionalSetpoint);
mxInit:= mxInit AND fbOffset8.mxInit(8,_wSDO2_OffsetsConditionalSetpoint);
END_METHOD

METHOD mxCollectInfoSDO3000 : BOOL
VAR_INPUT
	bIndex	: BYTE;
	rValue	: REAL;
END_VAR
mxCollectInfoSDO3000 := TRUE;
// Check index
IF bIndex <= 0 OR bIndex > bAmountOffsets THEN
	mxCollectInfoSDO3000 := FALSE;
	RETURN;
END_IF

adi_Testing[bIndex]:=TO_DINT(rValue);
END_METHOD

METHOD mxOD3000Define : BOOL
VAR_INPUT
	itf0D3000	: itf_od3000;
END_VAR
VAR
	Data		: _OD3000Struct_RegistrationData;
	bOffset		: BYTE := 28;
	i			: BYTE;
END_VAR
mxOD3000Define:=TRUE;

// Define SDO 3000
mxOD3000Define:=TRUE;
IF xActive THEN
	FOR i := 1 TO bAmountOffsets DO
		Data.wIndex		:= _wSDO3_STC_oilfree_Testing;
		Data.bSubIndex	:= i + bOffset;										 
		Data.pData		:= ADR(adi_Testing[i]);
		Data.wAttrib	:= _OD3000_wSubIndexRead;
		mxOD3000Define	:= mxOD3000Define AND itf0D3000.mxAdd(Data);
	END_FOR
END_IF
END_METHOD

METHOD mxRun : BOOL
VAR_INPUT
END_VAR
IF NOT xActive THEN
	RETURN;
END_IF

fbOffset1.mxGetInput();
mxCollectInfoSDO3000(1, fbOffset1.prprValue); 
fbOffset2.mxGetInput();
mxCollectInfoSDO3000(2, fbOffset2.prprValue);
fbOffset3.mxGetInput();
mxCollectInfoSDO3000(3, fbOffset3.prprValue);
fbOffset4.mxGetInput();
mxCollectInfoSDO3000(4, fbOffset4.prprValue);
fbOffset5.mxGetInput();
mxCollectInfoSDO3000(5, fbOffset5.prprValue);
fbOffset6.mxGetInput();
mxCollectInfoSDO3000(6, fbOffset6.prprValue);
fbOffset7.mxGetInput();
mxCollectInfoSDO3000(7, fbOffset7.prprValue);
fbOffset8.mxGetInput();
mxCollectInfoSDO3000(8, fbOffset8.prprValue);
END_METHOD

METHOD mxGetValueOffset : BOOL
VAR_INPUT
	bOffsetNumber		: BYTE;
END_VAR
VAR_OUTPUT
	rValue				: REAL;
END_VAR
mxGetValueOffset := TRUE;
CASE bOffsetNumber OF 
	1: rValue := fbOffset1.prprValue;
	
	2: rValue := fbOffset2.prprValue;
	
	3: rValue := fbOffset3.prprValue;
	
	4: rValue := fbOffset4.prprValue;
	
	5: rValue := fbOffset5.prprValue;
	
	6: rValue := fbOffset6.prprValue;
	
	7: rValue := fbOffset7.prprValue;
	
	8: rValue := fbOffset8.prprValue;
	
	ELSE
		mxGetValueOffset := FALSE;
END_CASE
END_METHOD

END_FUNCTION_BLOCK

// Oil Free Air/Offset/fbtOffset
FUNCTION_BLOCK fbtOffset
VAR	
	bInputNumber									: BYTE;
	xStatus											: BOOL := FALSE;
	
	itfLocalRoot									: itf_SystemRoot;
	bType											: BYTE:=ENUM_meas_internal_fixed.UNKNOWN;
	bCalculationType								: BYTE;
	sPowerValue										: SINT;
	
	itfMeasurement									: itf_baseio;
	itfIData										: itf_InternalValue;
	dwFixedValue									: DWORD;	
	dwSafetyValue									: DWORD;

	rValue											: REAL;	
	xZeroValue										: BOOL;
	_wSDO2_OffsetConditionalSetpointCalculation		: WORD;
	
END_VAR

(*
Stijn Staring - 31/03/23
This offset function should be used together with the Conditional Setpoint Calculation functions.
In the Conditional Setpoint Calculation functions there will be options provided to apply the offset. 

Options =>
•	Absolute offset: the obvious; add or substract the given value
•	IData
•	MPL

Safety value to detect a sensor error.
*)

PROPERTY prprValue : REAL
GET
prprValue:=rValue;
END_GET
END_PROPERTY

METHOD mxGetInput : BOOL
VAR_INPUT
END_VAR
VAR
	diValue_Tmp	: DINT;
	iMinRange	: INT;
	iMaxRange	: INT;
	wRange		: WORD;	
	TmpItem		: ODItem;
END_VAR
IF NOT xStatus THEN
		rValue :=0;
	RETURN;
END_IF

CASE bType OF 
	
	ENUM_meas_internal_fixed.MeasuredValue:
		IF NOT itfMeasurement.prpxSensorError THEN
			itfMeasurement.mxGetValueINT(iValueOut => diValue_Tmp);
			itfMeasurement.mxGetRanges(iMinRange=> iMinRange, iMaxRange=> iMaxRange,wRange=> wRange);
			rValue:=DINT_TO_REAL(LIMIT(iMinRange,diValue_Tmp, iMaxRange));
		ELSE
			rValue := DWORD_TO_REAL(dwSafetyValue);
		END_IF

	ENUM_meas_internal_fixed.InternalValue:
		itfIData.mxGetValueDINT( diValueOut => diValue_Tmp);
		rValue:=DINT_TO_REAL(diValue_Tmp);
		
	ENUM_meas_internal_fixed.FixedValue:
		CmpODRead(_wSDO2_OffsetConditionalSetpointCalculation, mxGetSubIndex(1), ADR(TmpItem));
		dwFixedValue:=TmpItem.dwValue;
		rValue:=DWORD_TO_REAL(dwFixedValue);	
		
END_CASE

// Check if Input is zero
xZeroValue:=FALSE;
IF rValue = 0 THEN
	xZeroValue:=TRUE;
END_IF

// Take sign into account
CASE bCalculationType OF
	0: 							//Add
 
	1: rvalue := -1 * rvalue;	//Subtract
	
END_CASE

// Apply power value
rvalue := TO_REAL(rvalue * EXPT(10, sPowerValue));
END_METHOD

METHOD mxInit : BOOL
VAR_INPUT
	bInputNumberIn	: BYTE;
	wSDO			: WORD;
END_VAR
VAR
	TmpItem		: ODItem;
	bOutputType	: BYTE;

END_VAR
mxInit:=TRUE;
bInputNumber:=bInputNumberIn;
_wSDO2_OffsetConditionalSetpointCalculation:=wSDO;

//Try to implement itfLocalRoot with SystemRoot of project
IF NOT __QUERYINTERFACE(GVL_itfRoot,itfLocalRoot) THEN
	mxInit:=FALSE;
	RETURN;
END_IF

IF NOT CmpODRead(_wSDO2_OffsetConditionalSetpointCalculation, mxGetSubIndex(3), ADR(TmpItem)) THEN
	rValue := 0;
	RETURN;
END_IF

bType:=TmpItem.bValue[1];
bCalculationType := TmpItem.bValue[2];
xStatus := BYTE_TO_BOOL(TmpItem.bValue[3]);

IF NOT xStatus THEN
	rValue :=0;
	RETURN;
END_IF

CmpODRead(_wSDO2_OffsetConditionalSetpointCalculation, mxGetSubIndex(2), ADR(TmpItem));

CASE bType OF 
	
	ENUM_meas_internal_fixed.MeasuredValue:
				IF TmpItem.wValue[1] = 0 THEN mxInit:= FALSE; RETURN; END_IF; 
				itfLocalRoot.prpitfLookupTables.prpitfMPLList.mxFind(wFind:=TmpItem.wValue[1], itfFound=>itfMeasurement); 		//Measurement		
				mxInit:=mxInit AND itfMeasurement<>0;
				
	ENUM_meas_internal_fixed.InternalValue:
		IF TmpItem.wValue[2] = 0 THEN mxInit:= FALSE; RETURN; END_IF; 
		itfLocalRoot.prpitfLookupTables.prpitfIVLList.mxFind(wFind:=TmpItem.wValue[2], itfFound=>itfIData);         // Internal variable
		mxInit:=mxInit AND itfIData<>0;
		
	ENUM_meas_internal_fixed.FixedValue:
		CmpODRead(_wSDO2_OffsetConditionalSetpointCalculation, mxGetSubIndex(1), ADR(TmpItem));
		dwFixedValue:=TmpItem.dwValue;			
			
	ELSE
		mxInit:=FALSE;
END_CASE

CmpODRead(_wSDO2_OffsetConditionalSetpointCalculation, mxGetSubIndex(4), ADR(TmpItem));
dwSafetyValue := TmpItem.dwValue;

// Reading in power value
mxGetPowerValue(sValue => sPowerValue);
END_METHOD

PROPERTY prpbInputNumber : BYTE
GET
prpbInputNumber:=bInputNumber;
END_GET
END_PROPERTY

METHOD mxGetSubIndex : BYTE
VAR_INPUT
	bOffset			: BYTE;
END_VAR
VAR
	bStartIndex					: BYTE:=0; //see Hi5
	bAmountOfSubIndicesForInput	: BYTE:=4; //see Hi5
END_VAR
mxGetSubIndex:= bStartIndex+bOffset+(bInputNumber-1)*bAmountOfSubIndicesForInput;
END_METHOD

PROPERTY prpxZeroValue : BOOL
GET
prpxZeroValue:=xZeroValue;
END_GET
END_PROPERTY

METHOD mxGetPowerValue : BOOL
VAR_INPUT
END_VAR
VAR_OUTPUT
	sValue				: SINT;
END_VAR
VAR
	bOffset 			: BYTE := 32;
	bSubIndex			: BYTE;
	bByteNumber			: BYTE;
	TmpItem				: ODItem;
END_VAR
IF bInputNumber <= 4 THEN
	bSubIndex := 1;
	bByteNumber := bInputNumber;
ELSIF bInputNumber <= 8 THEN
	bSubIndex := 2;
	bByteNumber := bInputNumber - 4;
END_IF
bSubIndex := bSubIndex + bOffset;

CmpODRead(_wSDO2_OffsetConditionalSetpointCalculation, bSubIndex, ADR(TmpItem));
sValue := TmpItem.sValue[bByteNumber];
END_METHOD

END_FUNCTION_BLOCK

// Handler/fbtSTCHandler
FUNCTION_BLOCK fbtSTCHandler IMPLEMENTS itf_STC_Handler
VAR
	fbEnergyRecoveryRegulation						: fbtEnergyRecoveryRegulation;
	fbOffsetsConditionalSetpointCalculation			: fbtOffsetsConditionalSetpointCalculation;
	
	fbConditionalSetpointCalculation1				: fbtConditionalSetpointCalculation;
	fbConditionalSetpointCalculation2				: fbtConditionalSetpointCalculation;
	fbConditionalSetpointCalculation3				: fbtConditionalSetpointCalculation;
	fbConditionalSetpointCalculation4				: fbtConditionalSetpointCalculation;
	fbConditionalSetpointCalculation5				: fbtConditionalSetpointCalculation;
	fbConditionalSetpointCalculation6				: fbtConditionalSetpointCalculation;
	
	fbOptimalSERCalculation							: fbtOptimalSERCalculation;
	
	bAmountOfValves									: BYTE := 6;
	afbAortaValves									: ARRAY[1..6] OF fbtAortaEngine_Base;
	awSTC_SDOs										: ARRAY[1..6] OF WORD := [16#27EB, 16#2958,  16#2959, 16#295A, 16#295B, 16#295C];
	awIVL_ActualPosition							: ARRAY[1..6] OF WORD := [13441, 13442, 13443, 13444, 13445, 13446];
	awIVL_ActualPosition_Name						: ARRAY[1..6] OF WORD := [gTxt_IDATA13441, gTxt_IDATA13442, gTxt_IDATA13443, gTxt_IDATA13444, gTxt_IDATA13445, gTxt_IDATA13446];
	awIVL_RequiredPosition							: ARRAY[1..6] OF WORD := [13447, 13448, 13449, 13450, 13451, 13452];
	awIVL_RequiredPosition_Name						: ARRAY[1..6] OF WORD := [gTxt_IDATA13447, gTxt_IDATA13448, gTxt_IDATA13449, gTxt_IDATA13450, gTxt_IDATA13451, gTxt_IDATA13452];
	

	
END_VAR

METHOD mxGetSTCValve : itf_STCValve
VAR_INPUT
	bNumber_STC	: BYTE;
END_VAR
VAR_OUTPUT
	
END_VAR
mxGetSTCValve := afbAortaValves[bNumber_STC];
END_METHOD

METHOD mxInit : BOOL
VAR_INPUT
	itfcondensationpointIn				: itf_condensationpoint;
END_VAR
VAR
	i	: int;
END_VAR
mxInit := TRUE;

mxInit := mxInit AND fbEnergyRecoveryRegulation.mxInit();
mxInit := mxInit AND fbOffsetsConditionalSetpointCalculation.mxInit();

mxInit := mxInit AND fbConditionalSetpointCalculation1.mxInit(_wSDO2_Conditional_Setpoint_Calculation1, fbEnergyRecoveryRegulation, itfcondensationpointIn, fbOffsetsConditionalSetpointCalculation);
mxInit := mxInit AND fbConditionalSetpointCalculation2.mxInit(_wSDO2_Conditional_Setpoint_Calculation2, fbEnergyRecoveryRegulation, itfcondensationpointIn, fbOffsetsConditionalSetpointCalculation);
mxInit := mxInit AND fbConditionalSetpointCalculation3.mxInit(_wSDO2_Conditional_Setpoint_Calculation3, fbEnergyRecoveryRegulation, itfcondensationpointIn, fbOffsetsConditionalSetpointCalculation);
mxInit := mxInit AND fbConditionalSetpointCalculation4.mxInit(_wSDO2_Conditional_Setpoint_Calculation4, fbEnergyRecoveryRegulation, itfcondensationpointIn, fbOffsetsConditionalSetpointCalculation);
mxInit := mxInit AND fbConditionalSetpointCalculation5.mxInit(_wSDO2_Conditional_Setpoint_Calculation5, fbEnergyRecoveryRegulation, itfcondensationpointIn, fbOffsetsConditionalSetpointCalculation);
mxInit := mxInit AND fbConditionalSetpointCalculation6.mxInit(_wSDO2_Conditional_Setpoint_Calculation6, fbEnergyRecoveryRegulation, itfcondensationpointIn, fbOffsetsConditionalSetpointCalculation);

mxInit := mxInit AND fbOptimalSERCalculation.mxInit(itfcondensationpointIn);

FOR i := 1 TO bAmountOfValves BY 1 DO
	mxInit := mxInit AND afbAortaValves[i].mxInit(awSTC_SDOs[i], itfEnergyRecoveryRegulationIn:=fbEnergyRecoveryRegulation);
END_FOR
END_METHOD

METHOD mxInit_Output : BOOL
VAR_INPUT
END_VAR
VAR
	i			: BYTE;
END_VAR
// mxInit_Output is needed next to a normal mxInit to make sure that the Idata is added to the list before it can be read out by another function. 

mxInit_Output := TRUE;

mxInit_Output := mxInit_Output AND fbEnergyRecoveryRegulation.mxInit_Output();

mxInit_Output := mxInit_Output AND fbConditionalSetpointCalculation1.mxInit_Output(_wSDO2_Conditional_Setpoint_Calculation1);
mxInit_Output := mxInit_Output AND fbConditionalSetpointCalculation2.mxInit_Output(_wSDO2_Conditional_Setpoint_Calculation2);
mxInit_Output := mxInit_Output AND fbConditionalSetpointCalculation3.mxInit_Output(_wSDO2_Conditional_Setpoint_Calculation2);
mxInit_Output := mxInit_Output AND fbConditionalSetpointCalculation4.mxInit_Output(_wSDO2_Conditional_Setpoint_Calculation4);
mxInit_Output := mxInit_Output AND fbConditionalSetpointCalculation5.mxInit_Output(_wSDO2_Conditional_Setpoint_Calculation5);
mxInit_Output := mxInit_Output AND fbConditionalSetpointCalculation6.mxInit_Output(_wSDO2_Conditional_Setpoint_Calculation6);

mxInit_Output := mxInit_Output AND fbOptimalSERCalculation.mxInit_Output();

FOR i := 1 TO bAmountOfValves BY 1 DO
	mxInit_Output := mxInit_Output AND afbAortaValves[i].mxInit_Output(i, awSTC_SDOs[i], awIVL_ActualPosition[i], awIVL_RequiredPosition[i], awIVL_ActualPosition_Name[i], awIVL_RequiredPosition_Name[i]);
END_FOR
END_METHOD

METHOD mxOD3000Define : BOOL
VAR_INPUT
	itf0D3000	: itf_od3000;
END_VAR
VAR
	i			: INT;
END_VAR
mxOD3000Define := TRUE;
mxOD3000Define := mxOD3000Define AND fbEnergyRecoveryRegulation.mxOD3000Define(itf0D3000);
mxOD3000Define := mxOD3000Define AND fbOffsetsConditionalSetpointCalculation.mxOD3000Define(itf0D3000);

mxOD3000Define := mxOD3000Define AND fbConditionalSetpointCalculation1.mxOD3000Define(itf0D3000);
mxOD3000Define := mxOD3000Define AND fbConditionalSetpointCalculation2.mxOD3000Define(itf0D3000);
mxOD3000Define := mxOD3000Define AND fbConditionalSetpointCalculation3.mxOD3000Define(itf0D3000);
mxOD3000Define := mxOD3000Define AND fbConditionalSetpointCalculation4.mxOD3000Define(itf0D3000);
mxOD3000Define := mxOD3000Define AND fbConditionalSetpointCalculation5.mxOD3000Define(itf0D3000);
mxOD3000Define := mxOD3000Define AND fbConditionalSetpointCalculation6.mxOD3000Define(itf0D3000);
FOR i := 1 TO bAmountOfValves BY 1 DO
	mxOD3000Define := mxOD3000Define AND afbAortaValves[i].mxOD3000Define(itf0D3000, awSTC_SDOs);
END_FOR
END_METHOD

METHOD mxRun : BOOL
VAR_INPUT
END_VAR
VAR
	i		: BYTE;
END_VAR
// Oil Free Air STC valve
fbEnergyRecoveryRegulation.mxRun();
fbOffsetsConditionalSetpointCalculation.mxRun();
fbConditionalSetpointCalculation1.mxRun();
fbConditionalSetpointCalculation2.mxRun();
fbConditionalSetpointCalculation3.mxRun();
fbConditionalSetpointCalculation4.mxRun();
fbConditionalSetpointCalculation5.mxRun();
fbConditionalSetpointCalculation6.mxRun();

// Industrial Air STC valve
fbOptimalSERCalculation.mRun();

// Generic STC valve
FOR i := 1 TO bAmountOfValves BY 1 DO
	afbAortaValves[i].mxRun();
END_FOR
END_METHOD

METHOD mxGetOptimalSERCalculation : itf_OptimalSERCalculation
VAR_INPUT
END_VAR
mxGetOptimalSERCalculation := fbOptimalSERCalculation;
END_METHOD

END_FUNCTION_BLOCK

// Oil Free Air/Energy Recovery Regulation/fbtEnergyRecoveryRegulation
FUNCTION_BLOCK fbtEnergyRecoveryRegulation IMPLEMENTS itf_EnergyRecoveryRegulation
VAR
	xActive							: BOOL;	
	bRequestMode					: BYTE;
	itfLocalRoot					: itf_SystemRoot;
	itf_RequestDigitalInput			: itf_baseio;
	fbWaterTempThreshold			: fbtInput_General;
	fbHeatQualityRef				: fbtInput_General;	
	bHeatQualityActive				: BYTE;
	iHeatQualityOffsetMinimal		: INT;
	iHeatQualityOffsetMedium		: INT;
	iHeatQualityOffsetMaximal		: INT;
	itf_HeatQualityOffsetIO			: itf_baseio;
	xHeatQualityOffsetIO_Possible	: BOOL;
	dwSafetyValueThreshold			: DWORD;
	
	bFlowSwitchInstalled			: BYTE;
	itf_FlowSwitch					: itf_baseio;
	xReverse						: BOOL;
	
	bWaterSensorInstalled			: BYTE;
	itf_WaterTemperature			: itf_baseio;
	iMaximumThreshold				: INT;
	iMinimumThreshold				: INT;
	
	xSwitch							: BOOL;
	
	fbIVL_ERSetpointTemp			: fbtIVL_ERSetpointTemp;
	rOutput							: REAL;
	diOutput_test					: DINT;
	dwTest1							: DWORD;
	dwTest2							: DWORD;

END_VAR

PROPERTY prprEnergyRecoverySetpointTemperature : REAL
GET
prprEnergyRecoverySetpointTemperature := rOutput;
END_GET
END_PROPERTY

METHOD mxInit : BOOL
VAR_INPUT
END_VAR
VAR
	TmpItem		: ODItem;
END_VAR
mxInit:=TRUE;
xActive:=TRUE;

IF NOT __QUERYINTERFACE(GVL_itfRoot,itfLocalRoot) THEN
	mxInit:=FALSE;
	RETURN;
END_IF

IF NOT CmpODRead(_wSDO2_EnergyRecoveryRegulation, 1 ,ADR(TmpItem)) THEN
	fbIVL_ERSetpointTemp.prpxDataBaseDefined := FALSE;
	xActive:=FALSE;
	RETURN;
END_IF

// Heat Quality
CmpODRead(_wSDO2_EnergyRecoveryRegulation, 1 ,ADR(TmpItem));
iHeatQualityOffsetMinimal := TmpItem.iValue[1];
iHeatQualityOffsetMedium := TmpItem.iValue[2];
CmpODRead(_wSDO2_EnergyRecoveryRegulation, 2 ,ADR(TmpItem));
iHeatQualityOffsetMaximal := TmpItem.iValue[1];
bHeatQualityActive := TmpItem.bValue[3];
mxInit:= mxInit AND fbHeatQualityRef.mxInit(3,_wSDO2_EnergyRecoveryRegulation, 0);

// bRequestMode = 0 => Display
// bRequestMode = 1 => Digital Input
bRequestMode := TmpItem.bValue[4];
CmpODRead(_wSDO2_EnergyRecoveryRegulation, 3 ,ADR(TmpItem));
IF TmpItem.wValue[1] = 0 THEN 
	bRequestMode := 0; 
ELSE
	itfLocalRoot.prpitfLookupTables.prpitfMPLList.mxFind(wFind:=TmpItem.wValue[1], itfFound=>itf_RequestDigitalInput); 		//Measurement		
	mxInit:=mxInit AND itf_RequestDigitalInput<>0;
END_IF

bFlowSwitchInstalled := TmpItem.bValue[3];
bWaterSensorInstalled := TmpItem.bValue[4];

CmpODRead(_wSDO2_EnergyRecoveryRegulation, 4 ,ADR(TmpItem));
IF BYTE_TO_BOOL(bFlowSwitchInstalled) THEN
	IF TmpItem.wValue[1] = 0 THEN 
		bFlowSwitchInstalled := 0; 
	ELSE
		itfLocalRoot.prpitfLookupTables.prpitfMPLList.mxFind(wFind:=TmpItem.wValue[1], itfFound=>itf_FlowSwitch); 		//Measurement		
		mxInit:=mxInit AND itf_FlowSwitch<>0;
	END_IF
END_IF

IF BYTE_TO_BOOL(bWaterSensorInstalled) THEN
	IF TmpItem.wValue[2] = 0 THEN 
		bWaterSensorInstalled := 0; 
	ELSE
		itfLocalRoot.prpitfLookupTables.prpitfMPLList.mxFind(wFind:=TmpItem.wValue[2], itfFound=>itf_WaterTemperature); 		//Measurement		
		mxInit:=mxInit AND itf_WaterTemperature<>0;
		mxInit:= mxInit AND fbWaterTempThreshold.mxInit(2,_wSDO2_EnergyRecoveryRegulation, 0);
	END_IF
END_IF

CmpODRead(_wSDO2_EnergyRecoveryRegulation, 9,ADR(TmpItem));
xReverse := BYTE_TO_BOOL(TmpItem.bValue[3]);

CmpODRead(_wSDO2_EnergyRecoveryRegulation, 19,ADR(TmpItem));
xHeatQualityOffsetIO_Possible := TRUE;
IF TmpItem.wValue[1] = 0 THEN 
	xHeatQualityOffsetIO_Possible := FALSE; 
ELSE
	itfLocalRoot.prpitfLookupTables.prpitfMPLList.mxFind(wFind:=TmpItem.wValue[1], itfFound=>itf_HeatQualityOffsetIO); 		//Measurement		
	mxInit:=mxInit AND itf_HeatQualityOffsetIO<>0;
END_IF

CmpODRead(_wSDO2_EnergyRecoveryRegulation, 20,ADR(TmpItem));
iMinimumThreshold := TmpItem.iValue[1];
iMaximumThreshold := TmpItem.iValue[2];

CmpODRead(_wSDO2_EnergyRecoveryRegulation, 22,ADR(TmpItem));
dwSafetyValueThreshold := TmpItem.dwValue;
END_METHOD

METHOD mxRun : BOOL
VAR_INPUT
END_VAR
VAR
	diTmpValue		: DINT;
	rTmpValue		: REAL;
	iMinRange		: INT;
	iMaxRange		: INT;
	wRange			: WORD;
	TmpItem			: ODItem;
END_VAR
IF NOT xActive THEN
	xSwitch := FALSE;
	RETURN;
END_IF

xSwitch := TRUE;
IF BYTE_TO_BOOL(bFlowSwitchInstalled) THEN
	IF xReverse THEN
		itf_FlowSwitch.mxGetValueINT(iValueOUt => diTmpValue);
		xSwitch := xSwitch AND NOT TO_BOOL(diTmpValue);
	ELSE
		itf_FlowSwitch.mxGetValueINT(iValueOUt => diTmpValue);
		xSwitch := xSwitch AND TO_BOOL(diTmpValue) AND NOT itf_FlowSwitch.prpxSensorError;
	END_IF
END_IF

IF BYTE_TO_BOOL(bWaterSensorInstalled) THEN
	itf_WaterTemperature.mxGetValueINT(iValueOut => diTmpValue);
	fbWaterTempThreshold.mxGetInput();
	IF iMinimumThreshold <> 0 OR iMaximumThreshold <> 0 THEN
		rTmpValue := LIMIT(iMinimumThreshold, fbWaterTempThreshold.prprValue, iMaximumThreshold);
	ELSE
		rTmpValue := fbWaterTempThreshold.prprValue;
	END_IF	
	xSwitch := xSwitch AND rTmpValue > TO_REAL(diTmpValue) AND NOT itf_WaterTemperature.prpxSensorError;
END_IF

CASE bRequestMode OF 
	// Display => still to be implemented
	0:	
	{warning Stijn: update THIS code, when display development is ready!}
		xSwitch := FALSE;
	// Digital Input
	1: 
		itf_RequestDigitalInput.mxGetValueINT(iValueOUt => diTmpValue);
		xSwitch := xSwitch AND TO_BOOL(diTmpValue);	
	ELSE
		xSwitch := FALSE;
END_CASE


IF bHeatQualityActive <> ENUM_HeatQualityOffset.Input_IO THEN
	fbHeatQualityRef.mxGetInput();
	rOutput := fbHeatQualityRef.prprValue;
END_IF	

// Heat Quality
CmpODRead(_wSDO2_EnergyRecoveryRegulation, 2 ,ADR(TmpItem));
bHeatQualityActive := TmpItem.bValue[3];

CASE bHeatQualityActive OF 

	ENUM_HeatQualityOffset.Input_IO:
		IF xHeatQualityOffsetIO_Possible THEN
			IF NOT itf_HeatQualityOffsetIO.prpxSensorError THEN
				itf_HeatQualityOffsetIO.mxGetValueINT(iValueOut => diTmpValue);
				itf_HeatQualityOffsetIO.mxGetRanges(iMinRange=> iMinRange, iMaxRange=> iMaxRange,wRange=> wRange);
				rOutput:=TO_REAL(LIMIT(iMinRange,diTmpValue, iMaxRange));
			ELSE
				rOutput := DWORD_TO_REAL(dwSafetyValueThreshold);
			END_IF
		ELSE
			bHeatQualityActive := ENUM_HeatQualityOffset.Not_used;
		END_IF 
		
	
	ENUM_HeatQualityOffset.Minimal:
		rOutput := rOutput + iHeatQualityOffsetMinimal;
		
	
	ENUM_HeatQualityOffset.Medium:
		rOutput := rOutput + iHeatQualityOffsetMedium;
		
	ENUM_HeatQualityOffset.Maximal:
		rOutput := rOutput + iHeatQualityOffsetMaximal;
		
END_CASE 

fbIVL_ERSetpointTemp.mxSetOutput(rOutput);

// Testing
diOutput_test := REAL_TO_DINT(rOutput);
dwTest1		  := bRequestMode;
dwTest2       := bHeatQualityActive;
END_METHOD

PROPERTY prpxSwitchToER : BOOL
GET
prpxSwitchToER := xSwitch;
END_GET
END_PROPERTY

METHOD mxOD3000Define : BOOL
VAR_INPUT
	itf0D3000	: itf_od3000;
END_VAR
VAR
	Data			: _OD3000Struct_RegistrationData;
END_VAR
mxOD3000Define:=TRUE;

// Define SDO 3000
IF xActive THEN
	
		Data.wIndex		:= _wSDO3_STC_oilfree_Testing;
		Data.bSubIndex	:= 87;										 
		Data.pData		:= ADR(diOutput_test);
		Data.wAttrib	:= _OD3000_wSubIndexRead;
		mxOD3000Define	:= mxOD3000Define AND itf0D3000.mxAdd(Data);
		
		Data.wIndex		:= _wSDO3_STC_oilfree_Testing;
		Data.bSubIndex	:= 88;										 
		Data.pData		:= ADR(dwTest1);
		Data.wAttrib	:= _OD3000_wSubIndexRead;
		mxOD3000Define	:= mxOD3000Define AND itf0D3000.mxAdd(Data);
		
		Data.wIndex		:= _wSDO3_STC_oilfree_Testing;
		Data.bSubIndex	:= 89;										 
		Data.pData		:= ADR(dwTest2);
		Data.wAttrib	:= _OD3000_wSubIndexRead;
		mxOD3000Define	:= mxOD3000Define AND itf0D3000.mxAdd(Data);		
		
END_IF
END_METHOD

METHOD mxInit_Output : BOOL
VAR_INPUT
END_VAR
VAR
	TmpItem		: ODItem;
END_VAR
mxInit_Output:=TRUE;
mxInit_Output:= mxInit_Output AND fbIVL_ERSetpointTemp.mxInit(_IVL_ER_Setpoint_Temperature);
END_METHOD

END_FUNCTION_BLOCK

// Oil Free Air/Energy Recovery Regulation/fbtIVL_ERSetpointTemp
FUNCTION_BLOCK fbtIVL_ERSetpointTemp EXTENDS fbtIVL_OutputBase
VAR
END_VAR

(*Stijn Staring - 05/04/2023*)

METHOD mxIVL_Settings_Overwrite : BOOL
VAR_INPUT
	wIVL_number	: WORD;
END_VAR
fbIVL_Out.mxInit(0, wIVL_number, _IVL_bAnalogType_Temperature);
END_METHOD

END_FUNCTION_BLOCK

// Oil Free Air/Conditional Setpoint/fbtConditionalSetpointCalculation
FUNCTION_BLOCK fbtConditionalSetpointCalculation
VAR
	xActive							: BOOL;
	xStatus_Condensation			: BOOL;
	xAuxProtectionActive			: BOOL;
	bNumber							: BYTE;
	_wSDO2_CondSetpoint				: WORD;
	fbUncond_Setpoint				: fbtInput_General;
	fbUpper_Limit_Setpoint			: fbtInput_General;
	fbLower_Limit_Setpoint			: fbtInput_General;
	fbAuxiliary_Temp				: fbtInput_General;
	fbERSetpoint					: fbtInput_CondSetpoint_ERSetpoint;
	fbIVL_CondSetpointTemp			: fbtIVL_CondSetpointTemp;
	itfcondensationpoint			: itf_condensationpoint;
	itfOffsets						: itf_OffsetsConditionalSetpointCalculation;
	iCondensationMinimum			: INT;
	iCondensationMaximum			: INT;
	// Conditional Setpoint SDOs
	awSDO							:  ARRAY[1..6] OF WORD := [_wSDO2_Conditional_Setpoint_Calculation1, _wSDO2_Conditional_Setpoint_Calculation2, _wSDO2_Conditional_Setpoint_Calculation3, _wSDO2_Conditional_Setpoint_Calculation4, _wSDO2_Conditional_Setpoint_Calculation5, _wSDO2_Conditional_Setpoint_Calculation6]; 
	// IVL numbers
	awIVL_numbers					: ARRAY[1..6] OF WORD := [_IVL_Conditional_Setpoint_Temperature_1, _IVL_Conditional_Setpoint_Temperature_2, _IVL_Conditional_Setpoint_Temperature_3, _IVL_Conditional_Setpoint_Temperature_4, _IVL_Conditional_Setpoint_Temperature_5, _IVL_Conditional_Setpoint_Temperature_6];
	// Testing
	adiTesting						: ARRAY[1..8] OF DINT;
	
END_VAR

(*
Stijn Staring - 05/04/2023
*)

METHOD mxInit : BOOL
VAR_INPUT
	wSDO								: WORD;
	itfEnergyRecoveryRegulationIn		: itf_EnergyRecoveryRegulation;
	itfcondensationpointIn				: itf_condensationpoint;
	itfOffsetsIn						: itf_OffsetsConditionalSetpointCalculation;
END_VAR
VAR
	TmpItem		: ODItem;
END_VAR
mxInit:=TRUE;
xActive:=TRUE;

_wSDO2_CondSetpoint:=wSDO;
IF NOT CmpODRead(_wSDO2_CondSetpoint, 1 ,ADR(TmpItem)) THEN
	fbIVL_CondSetpointTemp.prpxDataBaseDefined := FALSE;
	xActive:=FALSE;
	RETURN;
END_IF

CmpODRead(_wSDO2_CondSetpoint, 32 ,ADR(TmpItem));
xAuxProtectionActive := BYTE_TO_BOOL(TmpItem.bValue[3]);

mxInit:= mxInit AND fbUncond_Setpoint.mxInit(1,_wSDO2_CondSetpoint, 0);
mxInit:= mxInit AND fbUpper_Limit_Setpoint.mxInit(2,_wSDO2_CondSetpoint, 0);
mxInit:= mxInit AND fbLower_Limit_Setpoint.mxInit(3,_wSDO2_CondSetpoint, 0);
IF xAuxProtectionActive THEN
	mxInit:= mxInit AND fbAuxiliary_Temp.mxInit(4,_wSDO2_CondSetpoint, 0);
END_IF
mxInit:= mxInit AND fbERSetpoint.mxInit_ER(5,_wSDO2_CondSetpoint, itfEnergyRecoveryRegulationIn);

// Condensation Temperature
IF CmpODRead(_wSDO2_CondensationPointCalculation, 1 ,ADR(TmpItem)) THEN
	CmpODRead(_wSDO2_CondSetpoint, 30 ,ADR(TmpItem));
	iCondensationMaximum := TmpItem.iValue[1];
	iCondensationMinimum := TmpItem.iValue[2];
	itfcondensationpoint := itfcondensationpointIn;
	CmpODRead(_wSDO2_CondSetpoint, 29 ,ADR(TmpItem));
	xStatus_Condensation := BYTE_TO_BOOL(TmpItem.bValue[1]) AND itfcondensationpoint<> 0;
ELSE 
	xStatus_Condensation := FALSE;
END_IF

itfOffsets := itfOffsetsIn;
IF itfOffsets = 0 THEN
	mxInit := FALSE;
END_IF
END_METHOD

METHOD mxInit_Output : BOOL
VAR_INPUT
	wSDO		: WORD;
END_VAR
VAR
	TmpItem		: ODItem;
	j			: DINT;
END_VAR
mxInit_Output:=TRUE;

// Find number of Conditional Setpoint Calculation
FOR j := LOWER_BOUND(awSDO, 1) TO UPPER_BOUND(awSDO, 1) DO
	IF awSDO[j] = wSDO THEN
		bNumber := DINT_TO_BYTE(j);
		EXIT;
	END_IF
END_FOR

fbIVL_CondSetpointTemp.prpwSDO := wSDO;
mxInit_Output:= mxInit_Output AND fbIVL_CondSetpointTemp.mxInit(awIVL_numbers[j]);
END_METHOD

METHOD mxRun : BOOL
VAR_INPUT
END_VAR
VAR
	iCondensationTemperature	: INT := -9999;
	rUncond_Setpoint_Value		: REAL;
	rUpper_Limit_Setpoint_Value	: REAL;
	rLower_Limit_Setpoint_Value : REAL;
	rAuxiliary_Temp				: REAL;
	rERSetpoint					: REAL;
	rOffset						: REAL;
	xSwitch						: BOOL;
	rMinimum					: REAL;
	rMaximum					: REAL;
	rResult						: REAL;
	
END_VAR
IF NOT xActive THEN
	RETURN;
END_IF

// Condensation Temperature
IF itfcondensationpoint <> 0 AND xStatus_Condensation THEN
	IF iCondensationMinimum = 0 AND iCondensationMaximum = 0 THEN
		iCondensationTemperature := itfcondensationpoint.prpiPDP;
	ELSE
		iCondensationTemperature := LIMIT(iCondensationMinimum, itfcondensationpoint.prpiPDP, iCondensationMaximum);
	END_IF
END_IF

// Get Inputs
fbUncond_Setpoint.mxGetInput();
fbUpper_Limit_Setpoint.mxGetInput();
fbLower_Limit_Setpoint.mxGetInput();
IF xAuxProtectionActive THEN
	fbAuxiliary_Temp.mxGetInput();
END_IF
fbERSetpoint.mxGetInput();

itfOffsets.mxGetValueOffset(bOffsetNumber := fbUncond_Setpoint.prpbOffsetNumber, rValue => rOffset);
rUncond_Setpoint_Value := fbUncond_Setpoint.prprValue + rOffset;
itfOffsets.mxGetValueOffset(bOffsetNumber := fbUpper_Limit_Setpoint.prpbOffsetNumber, rValue => rOffset);
rUpper_Limit_Setpoint_Value := fbUpper_Limit_Setpoint.prprValue + rOffset;
itfOffsets.mxGetValueOffset(bOffsetNumber := fbLower_Limit_Setpoint.prpbOffsetNumber, rValue => rOffset);
rLower_Limit_Setpoint_Value := fbLower_Limit_Setpoint.prprValue + rOffset;
IF xAuxProtectionActive THEN
	itfOffsets.mxGetValueOffset(bOffsetNumber := fbAuxiliary_Temp.prpbOffsetNumber, rValue => rOffset);
	rAuxiliary_Temp := fbAuxiliary_Temp.prprValue + rOffset;
ELSE
	rAuxiliary_Temp := rUpper_Limit_Setpoint_Value;
END_IF
itfOffsets.mxGetValueOffset(bOffsetNumber := fbERSetpoint.prpbOffsetNumber, rValue => rOffset);
rERSetpoint := fbERSetpoint.prprValue + rOffset;

xSwitch := fbERSetpoint.prpxSwitchToER;

IF xSwitch AND fbERSetpoint.prpxStatus THEN
	
	rMinimum := MIN(rERSetpoint, rUpper_Limit_Setpoint_Value, rAuxiliary_Temp);
	
ELSE
	rMinimum := MIN(rUncond_Setpoint_Value, rUpper_Limit_Setpoint_Value, rAuxiliary_Temp);
END_IF

IF xStatus_Condensation THEN
	rMaximum := MAX(rMinimum, rLower_Limit_Setpoint_Value, iCondensationTemperature);
ELSE 
	rMaximum := MAX(rMinimum, rLower_Limit_Setpoint_Value);
END_IF

IF xSwitch AND fbERSetpoint.prpxStatus THEN	
	itfOffsets.mxGetValueOffset(bOffsetNumber := fbIVL_CondSetpointTemp.prpbOffsetNumberER, rValue => rOffset);
ELSE
	itfOffsets.mxGetValueOffset(bOffsetNumber := fbIVL_CondSetpointTemp.prpbOffsetNumber, rValue => rOffset);
END_IF
rResult := rMaximum + rOffset;

fbIVL_CondSetpointTemp.mxSetOutput(rResult);

// Testing
mxCollectInfoSDO3000(1, iCondensationTemperature);
mxCollectInfoSDO3000(2, fbUncond_Setpoint.prprValue);
mxCollectInfoSDO3000(3, fbUpper_Limit_Setpoint.prprValue);
mxCollectInfoSDO3000(4, fbLower_Limit_Setpoint.prprValue);
IF xAuxProtectionActive THEN
	mxCollectInfoSDO3000(5, fbAuxiliary_Temp.prprValue);
END_IF
mxCollectInfoSDO3000(6, fbERSetpoint.prprValue);
mxCollectInfoSDO3000(7, BOOL_TO_REAL(xSwitch));
mxCollectInfoSDO3000(8, rResult);
END_METHOD

METHOD mxOD3000Define : BOOL
VAR_INPUT
	itf0D3000	: itf_od3000;
END_VAR
VAR
	Data			: _OD3000Struct_RegistrationData;
	bOffset			: BYTE := 38;
	i				: BYTE;
	bAmountOfData	: BYTE;
END_VAR
mxOD3000Define:=TRUE;

bAmountOfData := TO_BYTE(SIZEOF(adiTesting));

// Define SDO 3000
IF xActive THEN
	FOR i := 1 TO bAmountOfData DO
		Data.wIndex		:= _wSDO3_STC_oilfree_Testing;
		Data.bSubIndex	:= i + bOffset + (bNumber - 1)*bAmountOfData;										 
		Data.pData		:= ADR(adiTesting[i]);
		Data.wAttrib	:= _OD3000_wSubIndexRead;
		mxOD3000Define	:= mxOD3000Define AND itf0D3000.mxAdd(Data);
	END_FOR
END_IF
END_METHOD

METHOD mxCollectInfoSDO3000 : BOOL
VAR_INPUT
	bIndex	: BYTE;
	rValue	: REAL;
END_VAR
mxCollectInfoSDO3000 := TRUE;
// Check index
IF bIndex <= 0 OR bIndex > TO_BYTE(SIZEOF(adiTesting)) THEN
	mxCollectInfoSDO3000 := FALSE;
	RETURN;
END_IF

adiTesting[bIndex]:=TO_DINT(rValue);
END_METHOD

END_FUNCTION_BLOCK

// Oil Free Air/Conditional Setpoint/fbtInput_CondSetpoint_ERSetpoint
FUNCTION_BLOCK fbtInput_CondSetpoint_ERSetpoint EXTENDS fbtInput_General
VAR
	itfEnergyRecoveryRegulation		:		itf_EnergyRecoveryRegulation;
	xSwitch							: 		BOOL;
END_VAR

(*Stijn Staring - 05/04/2023*)

METHOD mxInit_ER : BOOL
VAR_INPUT
	bInputNumberIn						: BYTE;
	wSDOIn								: WORD;
	itfEnergyRecoveryRegulationIn		:		itf_EnergyRecoveryRegulation;
END_VAR
VAR
	TmpItem		: ODItem;
	bOutputType	: BYTE;
END_VAR
mxInit_ER:=TRUE;
bInputNumber:=bInputNumberIn;
wSDO:=wSDOIn;

//Try to implement itfLocalRoot with SystemRoot of project
IF NOT __QUERYINTERFACE(GVL_itfRoot,itfLocalRoot) THEN
	mxInit_ER:=FALSE;
	RETURN;
END_IF

IF NOT CmpODRead(wSDO, mxGetSubIndex(3), ADR(TmpItem)) THEN
	xStatus := FALSE;
	rValue := 0;
	RETURN;
END_IF

itfEnergyRecoveryRegulation := itfEnergyRecoveryRegulationIn;
bType:=ENUM_meas_internal_fixed.InternalValue;	
bOffset := TmpItem.bValue[1];

CmpODRead(wSDO, mxGetSubIndex(5), ADR(TmpItem));
xStatus := BYTE_TO_BOOL(TmpItem.bValue[2]) AND CmpODRead(_wSDO2_EnergyRecoveryRegulation, 1 ,ADR(TmpItem));
IF xStatus AND itfEnergyRecoveryRegulationIn = 0 THEN
	mxInit_ER := FALSE;
END_IF
END_METHOD

METHOD mxGetInput : BOOL
IF NOT xStatus THEN
		rValue :=0;
	RETURN;
END_IF

rValue := itfEnergyRecoveryRegulation.prprEnergyRecoverySetpointTemperature;

IF itfEnergyRecoveryRegulation <> 0 THEN
	xSwitch :=itfEnergyRecoveryRegulation.prpxSwitchToER;
END_IF

// Check if Input is zero
xZeroValue:=FALSE;
IF rValue = 0 THEN
	xZeroValue:=TRUE;
END_IF
END_METHOD

PROPERTY prpxSwitchToER : BOOL
GET
prpxSwitchToER := xSwitch;
END_GET
END_PROPERTY

END_FUNCTION_BLOCK

// Oil Free Air/Conditional Setpoint/fbtIVL_CondSetpointTemp
FUNCTION_BLOCK fbtIVL_CondSetpointTemp EXTENDS fbtIVL_OutputBase
VAR
	bOffsetER				: BYTE;
	bOffset					: BYTE;
	iMinimumOutput			: INT;
	iMaximumOutput			: INT;
	wSDO					: WORD;
END_VAR

(*Stijn Staring - 05/04/2023*)

METHOD mxSetOutput : BOOL
VAR_INPUT
	rValue		: REAL;
END_VAR
VAR
	iMinRange	: INT;
	iMaxRange	: INT;
	wRange		: WORD;
END_VAR
mxSetOutput	:= FALSE;

IF iMinimumOutput <> 0 OR iMaximumOutput <> 0 THEN
	rValue := LIMIT(iMinimumOutput, rValue, iMaximumOutput);
END_IF

SUPER^.mxSetOutput(rValue);
END_METHOD

PROPERTY prpwSDO : WORD
SET
wSDO := prpwSDO;
END_SET
END_PROPERTY

METHOD mxInit : BOOL
VAR_INPUT
	wIVL_number		: WORD;
END_VAR
VAR
	TmpItem		: ODItem;
	bIVLType	: BYTE;
END_VAR
mxInit:=TRUE;
mxInit := SUPER^.mxInit(wIVL_number);			

CmpODRead(wSDO, 29, ADR(TmpItem));
bOffset   := TmpItem.bValue[3];
bOffsetER := TmpItem.bValue[4];

CmpODRead(wSDO, 31, ADR(TmpItem));
iMinimumOutput := TmpItem.iValue[1];
iMaximumOutput := TmpItem.iValue[2];
END_METHOD

PROPERTY prpbOffsetNumber : BYTE
GET
prpbOffsetNumber := bOffset;
END_GET
END_PROPERTY

PROPERTY prpbOffsetNumberER : BYTE
GET
prpbOffsetNumberER := bOffsetER;
END_GET
END_PROPERTY

METHOD mxIVL_Settings_Overwrite : BOOL
VAR_INPUT
	wIVL_number	: WORD;
END_VAR
fbIVL_Out.mxInit(0, wIVL_number, _IVL_bAnalogType_Temperature);
END_METHOD

END_FUNCTION_BLOCK

// Industrial Air SER Calculation/fbtOptimalSERCalculation
FUNCTION_BLOCK fbtOptimalSERCalculation IMPLEMENTS itf_OptimalSERCalculation
VAR	
	xActive	: BOOL	:= TRUE;

	itfSpeedControl		: itf_SpeedControl;
	itfConverterInfo	: itf_ConverterInfo;
	itfLookupTables		: itf_Lookuptables;
	
	itfAmbientAirTemperature	: itf_BaseIO;
	itfPressure					: itf_BaseIO;
	
	wA	: WORD;
	bB	: BYTE;
	bC	: BYTE;
	iD	: INT;
	bRegulationType		: BYTE;
	
	iTemperature	: INT;
	
	itfcondensationpoint				: itf_condensationpoint;
	
	// Idata
	fbIVL_OptimalSERTemp				: fbtIVL_OptimalSERTemp;
	fbIVL_OptimalSERTemp_Limited		: fbtIVL_OptimalSERTemp;
	
	// Debug
	xDebug				: BOOL	:= TRUE;
	diDebugTemperature	: DINT;
	
	fbRamp		: RAMP_REAL;
	rAscend		: REAL;
	rDescend	: REAL;
	tTimeBase	: TIME;
END_VAR

METHOD mxInit : BOOL
VAR_INPUT
	itfcondensationpointIn		: itf_condensationpoint;
END_VAR
VAR
	itfLocalRoot		: itf_SystemRoot;
	itfDrives			: itf_ConverterInterfaces;
	itfCompConverter	: itf_Converter;
	TmpItem	: ODItem;
END_VAR
mxInit := TRUE;

// Handle cases where this is not needed
IF NOT CmpODRead(ENUM_SDO_2000.OptimalSERCalculation,	1,	ADR(TmpItem)) THEN
	fbIVL_OptimalSERTemp.prpxDataBaseDefined 		 := FALSE;	
	fbIVL_OptimalSERTemp_Limited.prpxDataBaseDefined := FALSE;
	xActive	:= FALSE;
	RETURN;
END_IF

IF NOT __QUERYINTERFACE(GVL_itfRoot, itfLocalRoot) THEN	mxInit := FALSE;	RETURN;	END_IF

itfLookupTables	:= itfLocalRoot.prpitfLookupTables;

IF		itfLookupTables			= 0
THEN	mxInit := FALSE;	RETURN;	END_IF

mxInit	:= mxInit AND mxLoadSettings(); // Need to load here to know regulation type

itfcondensationpoint := itfcondensationpointIn;

	
IF bRegulationType = 11 THEN // VSD
	itfDrives		:= itfLocalRoot.prpitfDrives;							
	itfSpeedControl	:= itfLocalRoot.prpitfSpeedControl;
	
	IF		itfDrives				= 0
	OR		itfSpeedControl			= 0
	THEN	mxInit := FALSE;	RETURN;	END_IF
	
	itfCompConverter := itfDrives.prpitfFirstMainOrCompressor;
	IF itfCompConverter <> 0 THEN
		itfConverterInfo := itfCompConverter.prpitfInfo;
		IF itfConverterInfo = 0 THEN
			mxInit := FALSE;
		 END_IF
	ELSE
		mxInit := FALSE;
	END_IF
END_IF
END_METHOD

METHOD PRIVATE mxLoadSettings : BOOL
VAR
	TmpItem	: ODItem;
END_VAR
mxLoadSettings := TRUE;

CmpODRead(ENUM_SDO_2000.OptimalSERCalculation,	1,	ADR(TmpItem));
mxLoadSettings	:= mxLoadSettings AND_THEN itfLookupTables.prpitfMPLList.mxFindType(TmpItem.wValue[1],	_IO_bTypeAnalogIn,	itfFound => itfAmbientAirTemperature);
mxLoadSettings	:= mxLoadSettings AND_THEN itfLookupTables.prpitfMPLList.mxFindType(TmpItem.wValue[2],	_IO_bTypeAnalogIn,	itfFound => itfPressure);

CmpODRead(ENUM_SDO_2000.OptimalSERCalculation,	2,	ADR(TmpItem));
wA	:= TmpItem.wValue[1];
bB	:= TmpItem.bValue[3];
bC	:= TmpItem.bValue[4];

CmpODRead(ENUM_SDO_2000.OptimalSERCalculation,	3,	ADR(TmpItem));
iD	:= TmpItem.iValue[1];
bRegulationType		:= TmpItem.bValue[4]; // 1 - FS | 11 - VSD

CmpODRead(ENUM_SDO_2000.OptimalSERCalculation,	4,	ADR(TmpItem));
rAscend		:= TmpItem.wValue[2];
rDescend	:= TmpItem.wValue[1];

CmpODRead(ENUM_SDO_2000.OptimalSERCalculation,	5,	ADR(TmpItem));
tTimeBase	:= TmpItem.wValue[1] * T#1MS;
END_METHOD

METHOD mRun : INT
VAR
	wCurrentMainSpeed		: WORD;
	wMaximumMainSpeed		: WORD;
	iAmbientAirTemperature	: INT;
	diPressure				: DINT;
	
	rOptimalTemperature	: REAL;
END_VAR
IF	NOT xActive	THEN
	RETURN;
END_IF

IF bRegulationType = 11 THEN // VSD
	wCurrentMainSpeed	:= itfConverterInfo.prpwActualRPM;
	wMaximumMainSpeed	:= itfSpeedControl.prpwMaxRpm;
	rOptimalTemperature	:= TO_REAL(wA) * 0.001 * TO_REAL(wCurrentMainSpeed) / TO_REAL(wMaximumMainSpeed);		// 0.0001 * Speed %
END_IF

itfAmbientAirTemperature.mxGetValueINT(iValueOut => iAmbientAirTemperature);
itfPressure.mxGetValueDINT_Pressure_mBar(diValueOut => diPressure);

rOptimalTemperature	:= rOptimalTemperature + (TO_REAL(bB) * 0.01 * TO_REAL(iAmbientAirTemperature) * 0.1);	// + 0.001 * degrees C
rOptimalTemperature	:= rOptimalTemperature + (TO_REAL(bC) * 0.1 * TO_REAL(diPressure) * 0.001);				// + 0.1 * pressure Bar
rOptimalTemperature	:= rOptimalTemperature + TO_REAL(iD) * 0.1;													// + 0.1
rOptimalTemperature	:= rOptimalTemperature * 10;															// + 0.1 degrees C

fbRamp(	IN			:= rOptimalTemperature,
		ASCEND		:= rAscend,
		DESCEND		:= rDescend,
		TIMEBASE	:= tTimeBase,
		RESET		:= FALSE,
		OUT			=> rOptimalTemperature);

iTemperature	:= TO_INT(rOptimalTemperature); // Property

fbIVL_OptimalSERTemp.mxSetOutput(rOptimalTemperature);

IF	xDebug	THEN
	diDebugTemperature	:= TO_DINT(rOptimalTemperature); // Debug
END_IF

// The optimal temperature should not cause any condensation. 
IF itfcondensationpoint <> 0 THEN
	rOptimalTemperature := MAX(rOptimalTemperature, itfCondensationPoint.prpiPDP);
END_IF
fbIVL_OptimalSERTemp_Limited.mxSetOutput(rOptimalTemperature);
END_METHOD

PROPERTY prpiTemperature : INT
GET
prpiTemperature := iTemperature;
END_GET
END_PROPERTY

PROPERTY prppdiDebugTemperature : POINTER TO DINT
GET
prppdiDebugTemperature := ADR(diDebugTemperature);
END_GET
END_PROPERTY

METHOD mxInit_Output : BOOL
VAR_INPUT
END_VAR
mxInit_Output:=TRUE;
mxInit_Output:= mxInit_Output AND fbIVL_OptimalSERTemp.mxInit(_IVL_OilTemperatureForOptimalSER);
mxInit_Output := mxInit_Output AND fbIVL_OptimalSERTemp_Limited.mxInit(_IVL_OilTemperatureForOptimalSER_Limited);
END_METHOD

END_FUNCTION_BLOCK

// Industrial Air SER Calculation/fbtIVL_OptimalSERTemp
FUNCTION_BLOCK fbtIVL_OptimalSERTemp EXTENDS fbtIVL_OutputBase
VAR
END_VAR

(*Stijn Staring - 05/04/2023*)

METHOD mxIVL_Settings_Overwrite : BOOL
VAR_INPUT
	wIVL_number			: WORD;
END_VAR
fbIVL_Out.mxInit(0, wIVL_number, _IVL_bAnalogType_Temperature); //If name is not showing, the fxGetIVLText function should be updated
END_METHOD

END_FUNCTION_BLOCK
